# EPICS substitutions: src/makeBaseApp/top/pcdsEvrApp/archiveSrc/archive__APPNAME_.substitutions
#
# _APPNAME_ substitutions file
#

# Generate iocAdmin archive request
file archive_iocAdmin.template
{
	{
		# Hack till msi supports empty substitutions
		_FOOBAR_=_FOOBAR_
	}
}

# Generate EVR archive request
file archive_evr.template
{
	{
		# Hack till msi supports empty substitutions
		_FOOBAR_=_FOOBAR_
	}
}
